TYPE STRUCT_CM_Sensor :
STRUCT
	Output		: BOOL;
	Auto		: BOOL;
	Manueel		: BOOL;
	Tag			: STRING;
END_STRUCT
END_TYPE

(* stored: Version 1.1.0.1, ProductVersion 3.1.4024.12
   DUT STRUCT_CM_Sensor: Id {ec4f0070-8049-4742-88e0-f11e394f9bf1} *)
